{attribute 'qualified_only'}
VAR_GLOBAL
	RecipeTypeTestSt	: ST_DebugTcHmi;
END_VAR

(* stored: Version 1.1.0.1
   GVL GVL_Debug: Id {c06a63c8-ff2b-0a68-26c8-eb69575b945a} *)
